FUNCTION_BLOCK FB_Blink
VAR_INPUT
	tON,tOff:TIME;
END_VAR
VAR_OUTPUT
	output:BOOL;
END_VAR
VAR
	timer:ton;
END_VAR

timer(IN:=NOT timer.Q);
IF timer.Q THEN
	IF output THEN
		timer.PT:=tOff;
	ELSE
		timer.PT:=tOn;
	END_IF
	output:= NOT output;
END_IF

END_FUNCTION_BLOCK

(* stored: Version 1.1.0.1, ProductVersion 3.1.4024.12
   POU FB_Blink: Id {0bc433c8-47a5-4115-82b7-cc053487ff41}, SpecialFunc None *)
